% RSLogix 500 project door control system.RSS, saved by version 8.30.00.16 %
PROJECT "UNTITLED"    % processor: Bul.1763 MicroLogix 1100 Series B %

PROGRAM FILES
  LAD 2   4 rungs

DATA FILES
  O0 OUTPUT  4 elements
  I1 INPUT  6 elements
  S2 STATUS  66 elements
  B3 BINARY  1 elements
  T4 TIMER  1 elements
  C5 COUNTER  1 elements
  R6 CONTROL  1 elements
  N7 INTEGER  1 elements
  F8 FLOAT  1 elements

LADDER 2
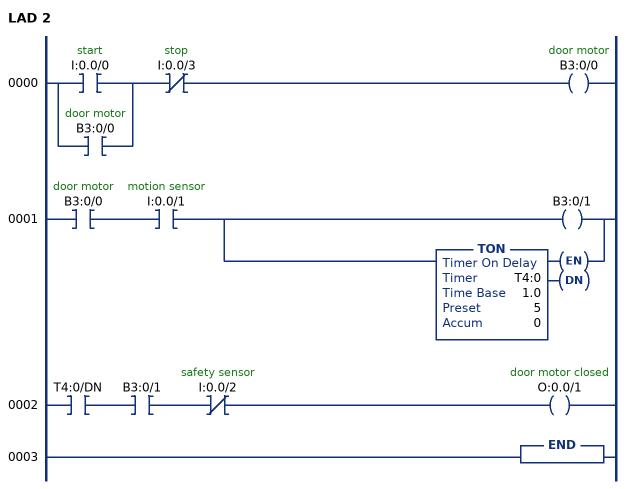
% Rung: 0 %
SOR BST XIC I:0.0/0 NXB XIC B3:0/0 BND XIO I:0.0/3 OTE B3:0/0 EOR
%   I:0.0/0  "start" %
%   B3:0/0  "door motor" %
%   I:0.0/3  "stop" %
% Rung: 1 %
SOR XIC B3:0/0 XIC I:0.0/1 BST OTE B3:0/1 NXB TON T4:0 1.0 5 0 BND EOR
%   B3:0/0  "door motor" %
%   I:0.0/1  "motion sensor" %
% Rung: 2 %
SOR XIC T4:0/DN XIC B3:0/1 XIO I:0.0/2 OTE O:0.0/1 EOR
%   I:0.0/2  "safety sensor" %
%   O:0.0/1  "door motor closed" %
% Rung: 3 %
SOR END EOR

OTHER DOCUMENTED ADDRESSES
  O:0.0/2  "door motor closed"

DATA TABLE (non-zero values as saved)
DATA B3
% B3:0 % 0X0001
DATA T4
% .PRE .ACC %
% T4:0 % 5 0
